Staubli VAL3: Cercle2.dtx

public frame fReference = {x=1500, y=200, z=-689.53, rz=90, fatherId=world[0]}
public jointRx jPark = {j3=90, j5=90}
public jointRx jJoint = {j1=-0.42016, j2=47.67737, j3=89.12207, j5=43.20056, j6=178.21616}
public mdesc mNomSpeed = {blend=off}
public mdesc mSpeed[6]
  [0] = {tmax=30, rmax=100, leave=0.1, reach=0.1, blend=cartesian}
  [1] = {tmax=30, rmax=100, leave=0.1, reach=0.1, blend=cartesian}
  [2] = {tmax=30, rmax=100, leave=0.1, reach=0.1, blend=cartesian}
  [3] = {tmax=30, rmax=100, leave=0.1, reach=0.1, blend=cartesian}
  [4] = {tmax=30, rmax=100, leave=0.1, reach=0.1, blend=cartesian}
  [5] = {tmax=30, rmax=100, leave=0.1, reach=0.1, blend=cartesian}
public num nTraj
num nTimeStop
num nTimeStart
num nMode
num nEtat
public pointRx pPoint[274]
  [0] = {x=-211, z=100, rx=-180, rz=88.636, shoulder=lefty, elbow=epositive, wrist=wpositive, fatherId=fReference[0]}
  [1] = {x=-211, rx=-180, rz=88.636, shoulder=lefty, elbow=epositive, wrist=wpositive, fatherId=fReference[0]}
  [2] = {x=-211, rx=-180, rz=88.636, shoulder=lefty, elbow=epositive, wrist=wpositive, fatherId=fReference[0]}
  [3] = {x=-210.761, y=-10.04, rx=-180, rz=85.909, shoulder=lefty, elbow=epositive, wrist=wpositive, fatherId=fReference[0]}
  [4] = {x=-210.045, y=-20.057, rx=-180, rz=83.182, shoulder=lefty, elbow=epositive, wrist=wpositive, fatherId=fReference[0]}
  [5] = {x=-208.852, y=-30.028, rx=-180, rz=80.455, shoulder=lefty, elbow=epositive, wrist=wpositive, fatherId=fReference[0]}
  [6] = {x=-207.187, y=-39.932, rx=-180, rz=77.727, shoulder=lefty, elbow=epositive, wrist=wpositive, fatherId=fReference[0]}
  [7] = {x=-205.052, y=-49.745, rx=-180, rz=75, shoulder=lefty, elbow=epositive, wrist=wpositive, fatherId=fReference[0]}
  [8] = {x=-202.453, y=-59.446, rx=-180, rz=72.273, shoulder=lefty, elbow=epositive, wrist=wpositive, fatherId=fReference[0]}
  [9] = {x=-199.395, y=-69.011, rx=-180, rz=69.545, shoulder=lefty, elbow=epositive, wrist=wpositive, fatherId=fReference[0]}
  [10] = {x=-195.886, y=-78.421, rx=-180, rz=66.818, shoulder=lefty, elbow=epositive, wrist=wpositive, fatherId=fReference[0]}
  [11] = {x=-191.932, y=-87.653, rx=-180, rz=64.091, shoulder=lefty, elbow=epositive, wrist=wpositive, fatherId=fReference[0]}
  [12] = {x=-187.544, y=-96.686, rx=-180, rz=61.364, shoulder=lefty, elbow=epositive, wrist=wpositive, fatherId=fReference[0]}
  [13] = {x=-182.731, y=-105.5, rx=180, rz=58.636, shoulder=lefty, elbow=epositive, wrist=wpositive, fatherId=fReference[0]}
  [14] = {x=-177.505, y=-114.075, rx=-180, rz=55.909, shoulder=lefty, elbow=epositive, wrist=wpositive, fatherId=fReference[0]}
  [15] = {x=-171.876, y=-122.392, rx=-180, rz=53.182, shoulder=lefty, elbow=epositive, wrist=wpositive, fatherId=fReference[0]}
  [16] = {x=-165.857, y=-130.432, rx=-180, rz=50.455, shoulder=lefty, elbow=epositive, wrist=wpositive, fatherId=fReference[0]}
  [17] = {x=-159.463, y=-138.176, rx=-180, rz=47.727, shoulder=lefty, elbow=epositive, wrist=wpositive, fatherId=fReference[0]}
  [18] = {x=-152.708, y=-145.607, rx=-180, rz=45, shoulder=lefty, elbow=epositive, wrist=wpositive, fatherId=fReference[0]}
  [19] = {x=-145.607, y=-152.708, rx=-180, rz=42.273, shoulder=lefty, elbow=epositive, wrist=wpositive, fatherId=fReference[0]}
  [20] = {x=-138.176, y=-159.463, rx=-180, rz=39.545, shoulder=lefty, elbow=epositive, wrist=wpositive, fatherId=fReference[0]}
  [21] = {x=-130.432, y=-165.857, rx=180, rz=36.818, shoulder=lefty, elbow=epositive, wrist=wpositive, fatherId=fReference[0]}
  [22] = {x=-122.392, y=-171.876, rx=180, rz=34.091, shoulder=lefty, elbow=epositive, wrist=wpositive, fatherId=fReference[0]}
  [23] = {x=-114.075, y=-177.505, rx=-180, rz=31.364, shoulder=lefty, elbow=epositive, wrist=wpositive, fatherId=fReference[0]}
  [24] = {x=-105.5, y=-182.731, rx=-180, rz=28.636, shoulder=lefty, elbow=epositive, wrist=wpositive, fatherId=fReference[0]}
  [25] = {x=-96.686, y=-187.544, rx=-180, rz=25.909, shoulder=lefty, elbow=epositive, wrist=wpositive, fatherId=fReference[0]}
  [26] = {x=-87.653, y=-191.932, rx=-180, rz=23.182, shoulder=lefty, elbow=epositive, wrist=wpositive, fatherId=fReference[0]}
  [27] = {x=-78.421, y=-195.886, rx=-180, rz=20.455, shoulder=lefty, elbow=epositive, wrist=wpositive, fatherId=fReference[0]}
  [28] = {x=-69.011, y=-199.395, rx=-180, rz=17.727, shoulder=lefty, elbow=epositive, wrist=wpositive, fatherId=fReference[0]}
  [29] = {x=-59.446, y=-202.453, rx=180, rz=15, shoulder=lefty, elbow=epositive, wrist=wpositive, fatherId=fReference[0]}
  [30] = {x=-49.745, y=-205.052, rx=180, rz=12.273, shoulder=lefty, elbow=epositive, wrist=wpositive, fatherId=fReference[0]}
  [31] = {x=-39.932, y=-207.187, rx=180, rz=9.545, shoulder=lefty, elbow=epositive, wrist=wpositive, fatherId=fReference[0]}
  [32] = {x=-30.028, y=-208.852, rx=-180, rz=6.818, shoulder=lefty, elbow=epositive, wrist=wpositive, fatherId=fReference[0]}
  [33] = {x=-20.057, y=-210.045, rx=-180, rz=4.091, shoulder=lefty, elbow=epositive, wrist=wpositive, fatherId=fReference[0]}
  [34] = {x=-10.04, y=-210.761, rx=180, rz=1.364, shoulder=lefty, elbow=epositive, wrist=wpositive, fatherId=fReference[0]}
  [35] = {y=-211, rx=180, rz=-1.364, shoulder=lefty, elbow=epositive, wrist=wpositive, fatherId=fReference[0]}
  [36] = {x=10.04, y=-210.761, rx=180, rz=-4.091, shoulder=lefty, elbow=epositive, wrist=wpositive, fatherId=fReference[0]}
  [37] = {x=20.057, y=-210.045, rx=-180, rz=-6.818, shoulder=lefty, elbow=epositive, wrist=wpositive, fatherId=fReference[0]}
  [38] = {x=30.028, y=-208.852, rx=180, rz=-9.545, shoulder=lefty, elbow=epositive, wrist=wpositive, fatherId=fReference[0]}
  [39] = {x=39.932, y=-207.187, rx=180, rz=-12.273, shoulder=lefty, elbow=epositive, wrist=wpositive, fatherId=fReference[0]}
  [40] = {x=49.745, y=-205.052, rx=-180, rz=-15, shoulder=lefty, elbow=epositive, wrist=wpositive, fatherId=fReference[0]}
  [41] = {x=59.446, y=-202.453, rx=-180, rz=-17.727, shoulder=lefty, elbow=epositive, wrist=wpositive, fatherId=fReference[0]}
  [42] = {x=69.011, y=-199.395, rx=180, rz=-20.455, shoulder=lefty, elbow=epositive, wrist=wpositive, fatherId=fReference[0]}
  [43] = {x=78.421, y=-195.886, rx=-180, rz=-23.182, shoulder=lefty, elbow=epositive, wrist=wpositive, fatherId=fReference[0]}
  [44] = {x=87.653, y=-191.932, rx=-180, rz=-25.909, shoulder=lefty, elbow=epositive, wrist=wpositive, fatherId=fReference[0]}
  [45] = {x=96.686, y=-187.544, rx=180, rz=-28.636, shoulder=lefty, elbow=epositive, wrist=wpositive, fatherId=fReference[0]}
  [46] = {x=105.5, y=-182.731, rx=-180, rz=-31.364, shoulder=lefty, elbow=epositive, wrist=wpositive, fatherId=fReference[0]}
  [47] = {x=114.075, y=-177.505, rx=180, rz=-34.091, shoulder=lefty, elbow=epositive, wrist=wpositive, fatherId=fReference[0]}
  [48] = {x=122.392, y=-171.876, rx=180, rz=-36.818, shoulder=lefty, elbow=epositive, wrist=wpositive, fatherId=fReference[0]}
  [49] = {x=130.432, y=-165.857, rx=180, rz=-39.545, shoulder=lefty, elbow=epositive, wrist=wpositive, fatherId=fReference[0]}
  [50] = {x=138.176, y=-159.463, rx=180, rz=-42.273, shoulder=lefty, elbow=epositive, wrist=wpositive, fatherId=fReference[0]}
  [51] = {x=145.607, y=-152.708, rx=180, rz=-45, shoulder=lefty, elbow=epositive, wrist=wpositive, fatherId=fReference[0]}
  [52] = {x=152.708, y=-145.607, rx=-180, rz=-47.727, shoulder=lefty, elbow=epositive, wrist=wpositive, fatherId=fReference[0]}
  [53] = {x=159.463, y=-138.176, rx=-180, rz=-50.455, shoulder=lefty, elbow=epositive, wrist=wpositive, fatherId=fReference[0]}
  [54] = {x=165.857, y=-130.432, rx=180, rz=-53.182, shoulder=lefty, elbow=epositive, wrist=wpositive, fatherId=fReference[0]}
  [55] = {x=171.876, y=-122.392, rx=-180, rz=-55.909, shoulder=lefty, elbow=epositive, wrist=wpositive, fatherId=fReference[0]}
  [56] = {x=177.505, y=-114.075, rx=180, rz=-58.636, shoulder=lefty, elbow=epositive, wrist=wpositive, fatherId=fReference[0]}
  [57] = {x=182.731, y=-105.5, rx=-180, rz=-61.364, shoulder=lefty, elbow=epositive, wrist=wpositive, fatherId=fReference[0]}
  [58] = {x=187.544, y=-96.686, rx=180, rz=-64.091, shoulder=lefty, elbow=epositive, wrist=wpositive, fatherId=fReference[0]}
  [59] = {x=191.932, y=-87.653, rx=180, rz=-66.818, shoulder=lefty, elbow=epositive, wrist=wpositive, fatherId=fReference[0]}
  [60] = {x=195.886, y=-78.421, rx=180, rz=-69.545, shoulder=lefty, elbow=epositive, wrist=wpositive, fatherId=fReference[0]}
  [61] = {x=199.395, y=-69.011, rx=180, rz=-72.273, shoulder=lefty, elbow=epositive, wrist=wpositive, fatherId=fReference[0]}
  [62] = {x=202.453, y=-59.446, rx=180, rz=-75, shoulder=lefty, elbow=epositive, wrist=wpositive, fatherId=fReference[0]}
  [63] = {x=205.052, y=-49.745, rx=180, rz=-77.727, shoulder=lefty, elbow=epositive, wrist=wpositive, fatherId=fReference[0]}
  [64] = {x=207.187, y=-39.932, rx=180, rz=-80.455, shoulder=lefty, elbow=epositive, wrist=wpositive, fatherId=fReference[0]}
  [65] = {x=208.852, y=-30.028, rx=180, rz=-83.182, shoulder=lefty, elbow=epositive, wrist=wpositive, fatherId=fReference[0]}
  [66] = {x=210.045, y=-20.057, rx=180, rz=-85.909, shoulder=lefty, elbow=epositive, wrist=wpositive, fatherId=fReference[0]}
  [67] = {x=210.761, y=-10.04, rx=180, rz=-88.636, shoulder=lefty, elbow=epositive, wrist=wpositive, fatherId=fReference[0]}
  [68] = {x=211, rx=-180, rz=-91.364, shoulder=lefty, elbow=epositive, wrist=wpositive, fatherId=fReference[0]}
  [69] = {x=210.761, y=10.04, rx=-180, rz=-94.091, shoulder=lefty, elbow=epositive, wrist=wpositive, fatherId=fReference[0]}
  [70] = {x=210.045, y=20.057, rx=-180, rz=-96.818, shoulder=lefty, elbow=epositive, wrist=wpositive, fatherId=fReference[0]}
  [71] = {x=208.852, y=30.028, rx=-180, rz=-99.545, shoulder=lefty, elbow=epositive, wrist=wpositive, fatherId=fReference[0]}
  [72] = {x=207.187, y=39.932, rx=-180, rz=-102.273, shoulder=lefty, elbow=epositive, wrist=wpositive, fatherId=fReference[0]}
  [73] = {x=205.052, y=49.745, rx=-180, rz=-105, shoulder=lefty, elbow=epositive, wrist=wpositive, fatherId=fReference[0]}
  [74] = {x=202.453, y=59.446, rx=-180, rz=-107.727, shoulder=lefty, elbow=epositive, wrist=wpositive, fatherId=fReference[0]}
  [75] = {x=199.395, y=69.011, rx=-180, rz=-110.455, shoulder=lefty, elbow=epositive, wrist=wpositive, fatherId=fReference[0]}
  [76] = {x=195.886, y=78.421, rx=-180, rz=-113.182, shoulder=lefty, elbow=epositive, wrist=wpositive, fatherId=fReference[0]}
  [77] = {x=191.932, y=87.653, rx=-180, rz=-115.909, shoulder=lefty, elbow=epositive, wrist=wpositive, fatherId=fReference[0]}
  [78] = {x=187.544, y=96.686, rx=-180, rz=-118.636, shoulder=lefty, elbow=epositive, wrist=wpositive, fatherId=fReference[0]}
  [79] = {x=182.731, y=105.5, rx=-180, rz=-121.364, shoulder=lefty, elbow=epositive, wrist=wpositive, fatherId=fReference[0]}
  [80] = {x=177.505, y=114.075, rx=-180, rz=-124.091, shoulder=lefty, elbow=epositive, wrist=wpositive, fatherId=fReference[0]}
  [81] = {x=171.876, y=122.392, rx=-180, rz=-126.818, shoulder=lefty, elbow=epositive, wrist=wpositive, fatherId=fReference[0]}
  [82] = {x=165.857, y=130.432, rx=-180, rz=-129.545, shoulder=lefty, elbow=epositive, wrist=wpositive, fatherId=fReference[0]}
  [83] = {x=159.463, y=138.176, rx=-180, rz=-132.273, shoulder=lefty, elbow=epositive, wrist=wpositive, fatherId=fReference[0]}
  [84] = {x=152.708, y=145.607, rx=-180, rz=-135, shoulder=lefty, elbow=epositive, wrist=wpositive, fatherId=fReference[0]}
  [85] = {x=145.607, y=152.708, rx=-180, rz=-137.727, shoulder=lefty, elbow=epositive, wrist=wpositive, fatherId=fReference[0]}
  [86] = {x=138.176, y=159.463, rx=-180, rz=-140.455, shoulder=lefty, elbow=epositive, wrist=wpositive, fatherId=fReference[0]}
  [87] = {x=130.432, y=165.857, rx=180, rz=-143.182, shoulder=lefty, elbow=epositive, wrist=wpositive, fatherId=fReference[0]}
  [88] = {x=122.392, y=171.876, rx=-180, rz=-145.909, shoulder=lefty, elbow=epositive, wrist=wpositive, fatherId=fReference[0]}
  [89] = {x=114.075, y=177.505, rx=-180, rz=-148.636, shoulder=lefty, elbow=epositive, wrist=wpositive, fatherId=fReference[0]}
  [90] = {x=105.5, y=182.731, rx=-180, rz=-151.364, shoulder=lefty, elbow=epositive, wrist=wpositive, fatherId=fReference[0]}
  [91] = {x=96.686, y=187.544, rx=-180, rz=-154.091, shoulder=lefty, elbow=epositive, wrist=wpositive, fatherId=fReference[0]}
  [92] = {x=87.653, y=191.932, rx=180, rz=-156.818, shoulder=lefty, elbow=epositive, wrist=wpositive, fatherId=fReference[0]}
  [93] = {x=78.421, y=195.886, rx=-180, rz=-159.545, shoulder=lefty, elbow=epositive, wrist=wpositive, fatherId=fReference[0]}
  [94] = {x=69.011, y=199.395, rx=180, rz=-162.273, shoulder=lefty, elbow=epositive, wrist=wpositive, fatherId=fReference[0]}
  [95] = {x=59.446, y=202.453, rx=-180, rz=-165, shoulder=lefty, elbow=epositive, wrist=wpositive, fatherId=fReference[0]}
  [96] = {x=49.745, y=205.052, rx=180, rz=-167.727, shoulder=lefty, elbow=epositive, wrist=wpositive, fatherId=fReference[0]}
  [97] = {x=39.932, y=207.187, rx=-180, rz=-170.455, shoulder=lefty, elbow=epositive, wrist=wpositive, fatherId=fReference[0]}
  [98] = {x=30.028, y=208.852, rx=-180, rz=-173.182, shoulder=lefty, elbow=epositive, wrist=wpositive, fatherId=fReference[0]}
  [99] = {x=20.057, y=210.045, rx=-180, rz=-175.909, shoulder=lefty, elbow=epositive, wrist=wpositive, fatherId=fReference[0]}
  [100] = {x=10.04, y=210.761, rx=-180, rz=-178.636, shoulder=lefty, elbow=epositive, wrist=wpositive, fatherId=fReference[0]}
  [101] = {y=211, rx=180, rz=178.636, shoulder=lefty, elbow=epositive, wrist=wpositive, fatherId=fReference[0]}
  [102] = {x=-10.04, y=210.761, rx=180, rz=175.909, shoulder=lefty, elbow=epositive, wrist=wpositive, fatherId=fReference[0]}
  [103] = {x=-20.057, y=210.045, rx=180, rz=173.182, shoulder=lefty, elbow=epositive, wrist=wpositive, fatherId=fReference[0]}
  [104] = {x=-30.028, y=208.852, rx=180, rz=170.455, shoulder=lefty, elbow=epositive, wrist=wpositive, fatherId=fReference[0]}
  [105] = {x=-39.932, y=207.187, rx=-180, rz=167.727, shoulder=lefty, elbow=epositive, wrist=wpositive, fatherId=fReference[0]}
  [106] = {x=-49.745, y=205.052, rx=-180, rz=165, shoulder=lefty, elbow=epositive, wrist=wpositive, fatherId=fReference[0]}
  [107] = {x=-59.446, y=202.453, rx=-180, rz=162.273, shoulder=lefty, elbow=epositive, wrist=wpositive, fatherId=fReference[0]}
  [108] = {x=-69.011, y=199.395, rx=-180, rz=159.545, shoulder=lefty, elbow=epositive, wrist=wpositive, fatherId=fReference[0]}
  [109] = {x=-78.421, y=195.886, rx=180, rz=156.818, shoulder=lefty, elbow=epositive, wrist=wpositive, fatherId=fReference[0]}
  [110] = {x=-87.653, y=191.932, rx=-180, rz=154.091, shoulder=lefty, elbow=epositive, wrist=wpositive, fatherId=fReference[0]}
  [111] = {x=-96.686, y=187.544, rx=180, rz=151.364, shoulder=lefty, elbow=epositive, wrist=wpositive, fatherId=fReference[0]}
  [112] = {x=-105.5, y=182.731, rx=-180, rz=148.636, shoulder=lefty, elbow=epositive, wrist=wpositive, fatherId=fReference[0]}
  [113] = {x=-114.075, y=177.505, rx=180, rz=145.909, shoulder=lefty, elbow=epositive, wrist=wpositive, fatherId=fReference[0]}
  [114] = {x=-122.392, y=171.876, rx=180, rz=143.182, shoulder=lefty, elbow=epositive, wrist=wpositive, fatherId=fReference[0]}
  [115] = {x=-130.432, y=165.857, rx=180, rz=140.455, shoulder=lefty, elbow=epositive, wrist=wpositive, fatherId=fReference[0]}
  [116] = {x=-138.176, y=159.463, rx=-180, rz=137.727, shoulder=lefty, elbow=epositive, wrist=wpositive, fatherId=fReference[0]}
  [117] = {x=-145.607, y=152.708, rx=180, rz=135, shoulder=lefty, elbow=epositive, wrist=wpositive, fatherId=fReference[0]}
  [118] = {x=-152.708, y=145.607, rx=180, rz=132.273, shoulder=lefty, elbow=epositive, wrist=wpositive, fatherId=fReference[0]}
  [119] = {x=-159.463, y=138.176, rx=180, rz=129.545, shoulder=lefty, elbow=epositive, wrist=wpositive, fatherId=fReference[0]}
  [120] = {x=-165.857, y=130.432, rx=180, rz=126.818, shoulder=lefty, elbow=epositive, wrist=wpositive, fatherId=fReference[0]}
  [121] = {x=-171.876, y=122.392, rx=180, rz=124.091, shoulder=lefty, elbow=epositive, wrist=wpositive, fatherId=fReference[0]}
  [122] = {x=-177.505, y=114.075, rx=180, rz=121.364, shoulder=lefty, elbow=epositive, wrist=wpositive, fatherId=fReference[0]}
  [123] = {x=-182.731, y=105.5, rx=180, rz=118.636, shoulder=lefty, elbow=epositive, wrist=wpositive, fatherId=fReference[0]}
  [124] = {x=-187.544, y=96.686, rx=180, rz=115.909, shoulder=lefty, elbow=epositive, wrist=wpositive, fatherId=fReference[0]}
  [125] = {x=-191.932, y=87.653, rx=180, rz=113.182, shoulder=lefty, elbow=epositive, wrist=wpositive, fatherId=fReference[0]}
  [126] = {x=-195.886, y=78.421, rx=180, rz=110.455, shoulder=lefty, elbow=epositive, wrist=wpositive, fatherId=fReference[0]}
  [127] = {x=-199.395, y=69.011, rx=180, rz=107.727, shoulder=lefty, elbow=epositive, wrist=wpositive, fatherId=fReference[0]}
  [128] = {x=-202.453, y=59.446, rx=180, rz=105, shoulder=lefty, elbow=epositive, wrist=wpositive, fatherId=fReference[0]}
  [129] = {x=-205.052, y=49.745, rx=180, rz=102.273, shoulder=lefty, elbow=epositive, wrist=wpositive, fatherId=fReference[0]}
  [130] = {x=-207.187, y=39.932, rx=180, rz=99.545, shoulder=lefty, elbow=epositive, wrist=wpositive, fatherId=fReference[0]}
  [131] = {x=-208.852, y=30.028, rx=180, rz=96.818, shoulder=lefty, elbow=epositive, wrist=wpositive, fatherId=fReference[0]}
  [132] = {x=-210.045, y=20.057, rx=180, rz=94.091, shoulder=lefty, elbow=epositive, wrist=wpositive, fatherId=fReference[0]}
  [133] = {x=-210.761, y=10.04, rx=180, rz=91.364, shoulder=lefty, elbow=epositive, wrist=wpositive, fatherId=fReference[0]}
  [134] = {x=-211, rx=180, rz=91.364, shoulder=lefty, elbow=epositive, wrist=wpositive, fatherId=fReference[0]}
  [135] = {x=-211, rx=180, rz=91.364, shoulder=lefty, elbow=epositive, wrist=wpositive, fatherId=fReference[0]}
  [136] = {x=-211, z=100, rx=180, rz=91.364, shoulder=lefty, elbow=epositive, wrist=wpositive, fatherId=fReference[0]}
  [137] = {x=-211, z=122, rx=180, rz=91.364, shoulder=lefty, elbow=epositive, wrist=wpositive, fatherId=fReference[0]}
  [138] = {x=-211, z=22, rx=180, rz=91.364, shoulder=lefty, elbow=epositive, wrist=wpositive, fatherId=fReference[0]}
  [139] = {x=-211, z=22, rx=180, rz=91.364, shoulder=lefty, elbow=epositive, wrist=wpositive, fatherId=fReference[0]}
  [140] = {x=-210.761, y=10.04, z=22, rx=180, rz=94.091, shoulder=lefty, elbow=epositive, wrist=wpositive, fatherId=fReference[0]}
  [141] = {x=-210.045, y=20.057, z=22, rx=180, rz=96.818, shoulder=lefty, elbow=epositive, wrist=wpositive, fatherId=fReference[0]}
  [142] = {x=-208.852, y=30.028, z=22, rx=180, rz=99.545, shoulder=lefty, elbow=epositive, wrist=wpositive, fatherId=fReference[0]}
  [143] = {x=-207.187, y=39.932, z=22, rx=180, rz=102.273, shoulder=lefty, elbow=epositive, wrist=wpositive, fatherId=fReference[0]}
  [144] = {x=-205.052, y=49.745, z=22, rx=180, rz=105, shoulder=lefty, elbow=epositive, wrist=wpositive, fatherId=fReference[0]}
  [145] = {x=-202.453, y=59.446, z=22, rx=180, rz=107.727, shoulder=lefty, elbow=epositive, wrist=wpositive, fatherId=fReference[0]}
  [146] = {x=-199.395, y=69.011, z=22, rx=180, rz=110.455, shoulder=lefty, elbow=epositive, wrist=wpositive, fatherId=fReference[0]}
  [147] = {x=-195.886, y=78.421, z=22, rx=-180, rz=113.182, shoulder=lefty, elbow=epositive, wrist=wpositive, fatherId=fReference[0]}
  [148] = {x=-191.932, y=87.653, z=22, rx=180, rz=115.909, shoulder=lefty, elbow=epositive, wrist=wpositive, fatherId=fReference[0]}
  [149] = {x=-187.544, y=96.686, z=22, rx=180, rz=118.636, shoulder=lefty, elbow=epositive, wrist=wpositive, fatherId=fReference[0]}
  [150] = {x=-182.731, y=105.5, z=22, rx=180, rz=121.364, shoulder=lefty, elbow=epositive, wrist=wpositive, fatherId=fReference[0]}
  [151] = {x=-177.505, y=114.075, z=22, rx=180, rz=124.091, shoulder=lefty, elbow=epositive, wrist=wpositive, fatherId=fReference[0]}
  [152] = {x=-171.876, y=122.392, z=22, rx=180, rz=126.818, shoulder=lefty, elbow=epositive, wrist=wpositive, fatherId=fReference[0]}
  [153] = {x=-165.857, y=130.432, z=22, rx=180, rz=129.545, shoulder=lefty, elbow=epositive, wrist=wpositive, fatherId=fReference[0]}
  [154] = {x=-159.463, y=138.176, z=22, rx=180, rz=132.273, shoulder=lefty, elbow=epositive, wrist=wpositive, fatherId=fReference[0]}
  [155] = {x=-152.708, y=145.607, z=22, rx=180, rz=135, shoulder=lefty, elbow=epositive, wrist=wpositive, fatherId=fReference[0]}
  [156] = {x=-145.607, y=152.708, z=22, rx=180, rz=137.727, shoulder=lefty, elbow=epositive, wrist=wpositive, fatherId=fReference[0]}
  [157] = {x=-138.176, y=159.463, z=22, rx=180, rz=140.455, shoulder=lefty, elbow=epositive, wrist=wpositive, fatherId=fReference[0]}
  [158] = {x=-130.432, y=165.857, z=22, rx=180, rz=143.182, shoulder=lefty, elbow=epositive, wrist=wpositive, fatherId=fReference[0]}
  [159] = {x=-122.392, y=171.876, z=22, rx=-180, rz=145.909, shoulder=lefty, elbow=epositive, wrist=wpositive, fatherId=fReference[0]}
  [160] = {x=-114.075, y=177.505, z=22, rx=180, rz=148.636, shoulder=lefty, elbow=epositive, wrist=wpositive, fatherId=fReference[0]}
  [161] = {x=-105.5, y=182.731, z=22, rx=180, rz=151.364, shoulder=lefty, elbow=epositive, wrist=wpositive, fatherId=fReference[0]}
  [162] = {x=-96.686, y=187.544, z=22, rx=180, rz=154.091, shoulder=lefty, elbow=epositive, wrist=wpositive, fatherId=fReference[0]}
  [163] = {x=-87.653, y=191.932, z=22, rx=-180, rz=156.818, shoulder=lefty, elbow=epositive, wrist=wpositive, fatherId=fReference[0]}
  [164] = {x=-78.421, y=195.886, z=22, rx=180, rz=159.545, shoulder=lefty, elbow=epositive, wrist=wpositive, fatherId=fReference[0]}
  [165] = {x=-69.011, y=199.395, z=22, rx=-180, rz=162.273, shoulder=lefty, elbow=epositive, wrist=wpositive, fatherId=fReference[0]}
  [166] = {x=-59.446, y=202.453, z=22, rx=-180, rz=165, shoulder=lefty, elbow=epositive, wrist=wpositive, fatherId=fReference[0]}
  [167] = {x=-49.745, y=205.052, z=22, rx=180, rz=167.727, shoulder=lefty, elbow=epositive, wrist=wpositive, fatherId=fReference[0]}
  [168] = {x=-39.932, y=207.187, z=22, rx=-180, rz=170.455, shoulder=lefty, elbow=epositive, wrist=wpositive, fatherId=fReference[0]}
  [169] = {x=-30.028, y=208.852, z=22, rx=180, rz=173.182, shoulder=lefty, elbow=epositive, wrist=wpositive, fatherId=fReference[0]}
  [170] = {x=-20.057, y=210.045, z=22, rx=-180, rz=175.909, shoulder=lefty, elbow=epositive, wrist=wpositive, fatherId=fReference[0]}
  [171] = {x=-10.04, y=210.761, z=22, rx=-180, rz=178.636, shoulder=lefty, elbow=epositive, wrist=wpositive, fatherId=fReference[0]}
  [172] = {y=211, z=22, rx=-180, rz=-178.636, shoulder=lefty, elbow=epositive, wrist=wpositive, fatherId=fReference[0]}
  [173] = {x=10.04, y=210.761, z=22, rx=180, rz=-175.909, shoulder=lefty, elbow=epositive, wrist=wpositive, fatherId=fReference[0]}
  [174] = {x=20.057, y=210.045, z=22, rx=-180, rz=-173.182, shoulder=lefty, elbow=epositive, wrist=wpositive, fatherId=fReference[0]}
  [175] = {x=30.028, y=208.852, z=22, rx=180, rz=-170.455, shoulder=lefty, elbow=epositive, wrist=wpositive, fatherId=fReference[0]}
  [176] = {x=39.932, y=207.187, z=22, rx=180, rz=-167.727, shoulder=lefty, elbow=epositive, wrist=wpositive, fatherId=fReference[0]}
  [177] = {x=49.745, y=205.052, z=22, rx=-180, rz=-165, shoulder=lefty, elbow=epositive, wrist=wpositive, fatherId=fReference[0]}
  [178] = {x=59.446, y=202.453, z=22, rx=-180, rz=-162.273, shoulder=lefty, elbow=epositive, wrist=wpositive, fatherId=fReference[0]}
  [179] = {x=69.011, y=199.395, z=22, rx=-180, rz=-159.545, shoulder=lefty, elbow=epositive, wrist=wpositive, fatherId=fReference[0]}
  [180] = {x=78.421, y=195.886, z=22, rx=180, rz=-156.818, shoulder=lefty, elbow=epositive, wrist=wpositive, fatherId=fReference[0]}
  [181] = {x=87.653, y=191.932, z=22, rx=180, rz=-154.091, shoulder=lefty, elbow=epositive, wrist=wpositive, fatherId=fReference[0]}
  [182] = {x=96.686, y=187.544, z=22, rx=-180, rz=-151.364, shoulder=lefty, elbow=epositive, wrist=wpositive, fatherId=fReference[0]}
  [183] = {x=105.5, y=182.731, z=22, rx=-180, rz=-148.636, shoulder=lefty, elbow=epositive, wrist=wpositive, fatherId=fReference[0]}
  [184] = {x=114.075, y=177.505, z=22, rx=-180, rz=-145.909, shoulder=lefty, elbow=epositive, wrist=wpositive, fatherId=fReference[0]}
  [185] = {x=122.392, y=171.876, z=22, rx=-180, rz=-143.182, shoulder=lefty, elbow=epositive, wrist=wpositive, fatherId=fReference[0]}
  [186] = {x=130.432, y=165.857, z=22, rx=-180, rz=-140.455, shoulder=lefty, elbow=epositive, wrist=wpositive, fatherId=fReference[0]}
  [187] = {x=138.176, y=159.463, z=22, rx=-180, rz=-137.727, shoulder=lefty, elbow=epositive, wrist=wpositive, fatherId=fReference[0]}
  [188] = {x=145.607, y=152.708, z=22, rx=-180, rz=-135, shoulder=lefty, elbow=epositive, wrist=wpositive, fatherId=fReference[0]}
  [189] = {x=152.708, y=145.607, z=22, rx=-180, rz=-132.273, shoulder=lefty, elbow=epositive, wrist=wpositive, fatherId=fReference[0]}
  [190] = {x=159.463, y=138.176, z=22, rx=-180, rz=-129.545, shoulder=lefty, elbow=epositive, wrist=wpositive, fatherId=fReference[0]}
  [191] = {x=165.857, y=130.432, z=22, rx=-180, rz=-126.818, shoulder=lefty, elbow=epositive, wrist=wpositive, fatherId=fReference[0]}
  [192] = {x=171.876, y=122.392, z=22, rx=-180, rz=-124.091, shoulder=lefty, elbow=epositive, wrist=wpositive, fatherId=fReference[0]}
  [193] = {x=177.505, y=114.075, z=22, rx=-180, rz=-121.364, shoulder=lefty, elbow=epositive, wrist=wpositive, fatherId=fReference[0]}
  [194] = {x=182.731, y=105.5, z=22, rx=-180, rz=-118.636, shoulder=lefty, elbow=epositive, wrist=wpositive, fatherId=fReference[0]}
  [195] = {x=187.544, y=96.686, z=22, rx=-180, rz=-115.909, shoulder=lefty, elbow=epositive, wrist=wpositive, fatherId=fReference[0]}
  [196] = {x=191.932, y=87.653, z=22, rx=-180, rz=-113.182, shoulder=lefty, elbow=epositive, wrist=wpositive, fatherId=fReference[0]}
  [197] = {x=195.886, y=78.421, z=22, rx=-180, rz=-110.455, shoulder=lefty, elbow=epositive, wrist=wpositive, fatherId=fReference[0]}
  [198] = {x=199.395, y=69.011, z=22, rx=-180, rz=-107.727, shoulder=lefty, elbow=epositive, wrist=wpositive, fatherId=fReference[0]}
  [199] = {x=202.453, y=59.446, z=22, rx=-180, rz=-105, shoulder=lefty, elbow=epositive, wrist=wpositive, fatherId=fReference[0]}
  [200] = {x=205.052, y=49.745, z=22, rx=-180, rz=-102.273, shoulder=lefty, elbow=epositive, wrist=wpositive, fatherId=fReference[0]}
  [201] = {x=207.187, y=39.932, z=22, rx=-180, rz=-99.545, shoulder=lefty, elbow=epositive, wrist=wpositive, fatherId=fReference[0]}
  [202] = {x=208.852, y=30.028, z=22, rx=-180, rz=-96.818, shoulder=lefty, elbow=epositive, wrist=wpositive, fatherId=fReference[0]}
  [203] = {x=210.045, y=20.057, z=22, rx=-180, rz=-94.091, shoulder=lefty, elbow=epositive, wrist=wpositive, fatherId=fReference[0]}
  [204] = {x=210.761, y=10.04, z=22, rx=-180, rz=-91.364, shoulder=lefty, elbow=epositive, wrist=wpositive, fatherId=fReference[0]}
  [205] = {x=211, z=22, rx=180, rz=-88.636, shoulder=lefty, elbow=epositive, wrist=wpositive, fatherId=fReference[0]}
  [206] = {x=210.761, y=-10.04, z=22, rx=180, rz=-85.909, shoulder=lefty, elbow=epositive, wrist=wpositive, fatherId=fReference[0]}
  [207] = {x=210.045, y=-20.057, z=22, rx=180, rz=-83.182, shoulder=lefty, elbow=epositive, wrist=wpositive, fatherId=fReference[0]}
  [208] = {x=208.852, y=-30.028, z=22, rx=180, rz=-80.455, shoulder=lefty, elbow=epositive, wrist=wpositive, fatherId=fReference[0]}
  [209] = {x=207.187, y=-39.932, z=22, rx=180, rz=-77.727, shoulder=lefty, elbow=epositive, wrist=wpositive, fatherId=fReference[0]}
  [210] = {x=205.052, y=-49.745, z=22, rx=180, rz=-75, shoulder=lefty, elbow=epositive, wrist=wpositive, fatherId=fReference[0]}
  [211] = {x=202.453, y=-59.446, z=22, rx=180, rz=-72.273, shoulder=lefty, elbow=epositive, wrist=wpositive, fatherId=fReference[0]}
  [212] = {x=199.395, y=-69.011, z=22, rx=180, rz=-69.545, shoulder=lefty, elbow=epositive, wrist=wpositive, fatherId=fReference[0]}
  [213] = {x=195.886, y=-78.421, z=22, rx=180, rz=-66.818, shoulder=lefty, elbow=epositive, wrist=wpositive, fatherId=fReference[0]}
  [214] = {x=191.932, y=-87.653, z=22, rx=180, rz=-64.091, shoulder=lefty, elbow=epositive, wrist=wpositive, fatherId=fReference[0]}
  [215] = {x=187.544, y=-96.686, z=22, rx=-180, rz=-61.364, shoulder=lefty, elbow=epositive, wrist=wpositive, fatherId=fReference[0]}
  [216] = {x=182.731, y=-105.5, z=22, rx=-180, rz=-58.636, shoulder=lefty, elbow=epositive, wrist=wpositive, fatherId=fReference[0]}
  [217] = {x=177.505, y=-114.075, z=22, rx=180, rz=-55.909, shoulder=lefty, elbow=epositive, wrist=wpositive, fatherId=fReference[0]}
  [218] = {x=171.876, y=-122.392, z=22, rx=180, rz=-53.182, shoulder=lefty, elbow=epositive, wrist=wpositive, fatherId=fReference[0]}
  [219] = {x=165.857, y=-130.432, z=22, rx=180, rz=-50.455, shoulder=lefty, elbow=epositive, wrist=wpositive, fatherId=fReference[0]}
  [220] = {x=159.463, y=-138.176, z=22, rx=180, rz=-47.727, shoulder=lefty, elbow=epositive, wrist=wpositive, fatherId=fReference[0]}
  [221] = {x=152.708, y=-145.607, z=22, rx=180, rz=-45, shoulder=lefty, elbow=epositive, wrist=wpositive, fatherId=fReference[0]}
  [222] = {x=145.607, y=-152.708, z=22, rx=180, rz=-42.273, shoulder=lefty, elbow=epositive, wrist=wpositive, fatherId=fReference[0]}
  [223] = {x=138.176, y=-159.463, z=22, rx=180, rz=-39.545, shoulder=lefty, elbow=epositive, wrist=wpositive, fatherId=fReference[0]}
  [224] = {x=130.432, y=-165.857, z=22, rx=180, rz=-36.818, shoulder=lefty, elbow=epositive, wrist=wpositive, fatherId=fReference[0]}
  [225] = {x=122.392, y=-171.876, z=22, rx=-180, rz=-34.091, shoulder=lefty, elbow=epositive, wrist=wpositive, fatherId=fReference[0]}
  [226] = {x=114.075, y=-177.505, z=22, rx=180, rz=-31.364, shoulder=lefty, elbow=epositive, wrist=wpositive, fatherId=fReference[0]}
  [227] = {x=105.5, y=-182.731, z=22, rx=180, rz=-28.636, shoulder=lefty, elbow=epositive, wrist=wpositive, fatherId=fReference[0]}
  [228] = {x=96.686, y=-187.544, z=22, rx=-180, rz=-25.909, shoulder=lefty, elbow=epositive, wrist=wpositive, fatherId=fReference[0]}
  [229] = {x=87.653, y=-191.932, z=22, rx=-180, rz=-23.182, shoulder=lefty, elbow=epositive, wrist=wpositive, fatherId=fReference[0]}
  [230] = {x=78.421, y=-195.886, z=22, rx=180, rz=-20.455, shoulder=lefty, elbow=epositive, wrist=wpositive, fatherId=fReference[0]}
  [231] = {x=69.011, y=-199.395, z=22, rx=180, rz=-17.727, shoulder=lefty, elbow=epositive, wrist=wpositive, fatherId=fReference[0]}
  [232] = {x=59.446, y=-202.453, z=22, rx=180, rz=-15, shoulder=lefty, elbow=epositive, wrist=wpositive, fatherId=fReference[0]}
  [233] = {x=49.745, y=-205.052, z=22, rx=180, rz=-12.273, shoulder=lefty, elbow=epositive, wrist=wpositive, fatherId=fReference[0]}
  [234] = {x=39.932, y=-207.187, z=22, rx=-180, rz=-9.545, shoulder=lefty, elbow=epositive, wrist=wpositive, fatherId=fReference[0]}
  [235] = {x=30.028, y=-208.852, z=22, rx=-180, rz=-6.818, shoulder=lefty, elbow=epositive, wrist=wpositive, fatherId=fReference[0]}
  [236] = {x=20.057, y=-210.045, z=22, rx=-180, rz=-4.091, shoulder=lefty, elbow=epositive, wrist=wpositive, fatherId=fReference[0]}
  [237] = {x=10.04, y=-210.761, z=22, rx=-180, rz=-1.364, shoulder=lefty, elbow=epositive, wrist=wpositive, fatherId=fReference[0]}
  [238] = {y=-211, z=22, rx=-180, rz=1.364, shoulder=lefty, elbow=epositive, wrist=wpositive, fatherId=fReference[0]}
  [239] = {x=-10.04, y=-210.761, z=22, rx=-180, rz=4.091, shoulder=lefty, elbow=epositive, wrist=wpositive, fatherId=fReference[0]}
  [240] = {x=-20.057, y=-210.045, z=22, rx=180, rz=6.818, shoulder=lefty, elbow=epositive, wrist=wpositive, fatherId=fReference[0]}
  [241] = {x=-30.028, y=-208.852, z=22, rx=-180, rz=9.545, shoulder=lefty, elbow=epositive, wrist=wpositive, fatherId=fReference[0]}
  [242] = {x=-39.932, y=-207.187, z=22, rx=-180, rz=12.273, shoulder=lefty, elbow=epositive, wrist=wpositive, fatherId=fReference[0]}
  [243] = {x=-49.745, y=-205.052, z=22, rx=180, rz=15, shoulder=lefty, elbow=epositive, wrist=wpositive, fatherId=fReference[0]}
  [244] = {x=-59.446, y=-202.453, z=22, rx=180, rz=17.727, shoulder=lefty, elbow=epositive, wrist=wpositive, fatherId=fReference[0]}
  [245] = {x=-69.011, y=-199.395, z=22, rx=-180, rz=20.455, shoulder=lefty, elbow=epositive, wrist=wpositive, fatherId=fReference[0]}
  [246] = {x=-78.421, y=-195.886, z=22, rx=-180, rz=23.182, shoulder=lefty, elbow=epositive, wrist=wpositive, fatherId=fReference[0]}
  [247] = {x=-87.653, y=-191.932, z=22, rx=-180, rz=25.909, shoulder=lefty, elbow=epositive, wrist=wpositive, fatherId=fReference[0]}
  [248] = {x=-96.686, y=-187.544, z=22, rx=-180, rz=28.636, shoulder=lefty, elbow=epositive, wrist=wpositive, fatherId=fReference[0]}
  [249] = {x=-105.5, y=-182.731, z=22, rx=-180, rz=31.364, shoulder=lefty, elbow=epositive, wrist=wpositive, fatherId=fReference[0]}
  [250] = {x=-114.075, y=-177.505, z=22, rx=-180, rz=34.091, shoulder=lefty, elbow=epositive, wrist=wpositive, fatherId=fReference[0]}
  [251] = {x=-122.392, y=-171.876, z=22, rx=180, rz=36.818, shoulder=lefty, elbow=epositive, wrist=wpositive, fatherId=fReference[0]}
  [252] = {x=-130.432, y=-165.857, z=22, rx=-180, rz=39.545, shoulder=lefty, elbow=epositive, wrist=wpositive, fatherId=fReference[0]}
  [253] = {x=-138.176, y=-159.463, z=22, rx=-180, rz=42.273, shoulder=lefty, elbow=epositive, wrist=wpositive, fatherId=fReference[0]}
  [254] = {x=-145.607, y=-152.708, z=22, rx=-180, rz=45, shoulder=lefty, elbow=epositive, wrist=wpositive, fatherId=fReference[0]}
  [255] = {x=-152.708, y=-145.607, z=22, rx=-180, rz=47.727, shoulder=lefty, elbow=epositive, wrist=wpositive, fatherId=fReference[0]}
  [256] = {x=-159.463, y=-138.176, z=22, rx=-180, rz=50.455, shoulder=lefty, elbow=epositive, wrist=wpositive, fatherId=fReference[0]}
  [257] = {x=-165.857, y=-130.432, z=22, rx=-180, rz=53.182, shoulder=lefty, elbow=epositive, wrist=wpositive, fatherId=fReference[0]}
  [258] = {x=-171.876, y=-122.392, z=22, rx=-180, rz=55.909, shoulder=lefty, elbow=epositive, wrist=wpositive, fatherId=fReference[0]}
  [259] = {x=-177.505, y=-114.075, z=22, rx=-180, rz=58.636, shoulder=lefty, elbow=epositive, wrist=wpositive, fatherId=fReference[0]}
  [260] = {x=-182.731, y=-105.5, z=22, rx=-180, rz=61.364, shoulder=lefty, elbow=epositive, wrist=wpositive, fatherId=fReference[0]}
  [261] = {x=-187.544, y=-96.686, z=22, rx=-180, rz=64.091, shoulder=lefty, elbow=epositive, wrist=wpositive, fatherId=fReference[0]}
  [262] = {x=-191.932, y=-87.653, z=22, rx=-180, rz=66.818, shoulder=lefty, elbow=epositive, wrist=wpositive, fatherId=fReference[0]}
  [263] = {x=-195.886, y=-78.421, z=22, rx=-180, rz=69.545, shoulder=lefty, elbow=epositive, wrist=wpositive, fatherId=fReference[0]}
  [264] = {x=-199.395, y=-69.011, z=22, rx=-180, rz=72.273, shoulder=lefty, elbow=epositive, wrist=wpositive, fatherId=fReference[0]}
  [265] = {x=-202.453, y=-59.446, z=22, rx=-180, rz=75, shoulder=lefty, elbow=epositive, wrist=wpositive, fatherId=fReference[0]}
  [266] = {x=-205.052, y=-49.745, z=22, rx=-180, rz=77.727, shoulder=lefty, elbow=epositive, wrist=wpositive, fatherId=fReference[0]}
  [267] = {x=-207.187, y=-39.932, z=22, rx=-180, rz=80.455, shoulder=lefty, elbow=epositive, wrist=wpositive, fatherId=fReference[0]}
  [268] = {x=-208.852, y=-30.028, z=22, rx=-180, rz=83.182, shoulder=lefty, elbow=epositive, wrist=wpositive, fatherId=fReference[0]}
  [269] = {x=-210.045, y=-20.057, z=22, rx=-180, rz=85.909, shoulder=lefty, elbow=epositive, wrist=wpositive, fatherId=fReference[0]}
  [270] = {x=-210.761, y=-10.04, z=22, rx=-180, rz=88.636, shoulder=lefty, elbow=epositive, wrist=wpositive, fatherId=fReference[0]}
  [271] = {x=-211, z=22, rx=-180, rz=88.636, shoulder=lefty, elbow=epositive, wrist=wpositive, fatherId=fReference[0]}
  [272] = {x=-211, z=22, rx=-180, rz=88.636, shoulder=lefty, elbow=epositive, wrist=wpositive, fatherId=fReference[0]}
  [273] = {x=-211, z=122, rx=-180, rz=88.636, shoulder=lefty, elbow=epositive, wrist=wpositive, fatherId=fReference[0]}
public tool tTool = {z=452, fatherId=flange[0], ioLink=valve1}
dio doValve1 = {link=valve1}
aio Tpompe = {link=CanIO\RemIO\remio0_QW}
